// TIA Portal project "Esercizio_contatore" (V15.1)

(* hardware
DEVICE "S7-1200 station_1"  S7-1200 Station
   slot 0: "Telaio di montaggio_0"  S7-1200 Rack  Rack  V1.0
   slot 1: "PLC_1"  CPU 1214C DC/DC/DC  6ES7 214-1AG40-0XB0  V4.2
*)

// ===== PLC "PLC_1"  CPU 1214C DC/DC/DC =====

VAR_GLOBAL CONSTANT   // PLC tag table "Tabella delle variabili standard"
   "valoreMassimo" : Int := 10;
END_VAR

DATA_BLOCK "blocco dati"   // DB1
{ S7_Optimized_Access := 'TRUE' }
VERSION : 0.1
   VAR RETAIN
      "A" : Array[0..9] of Int;
      contatore : Int;
   END_VAR
BEGIN
END_DATA_BLOCK

ORGANIZATION_BLOCK "Main"   // OB1, LAD, ProgramCycle
TITLE = "Main Program Sweep (Cycle)"
{ S7_Optimized_Access := 'TRUE' }
VERSION : 0.1
   VAR_INPUT
      Initial_Call : Bool;   // Initial call of this OB
      Remanence : Bool;   // =True, if remanent data are available
   END_VAR
BEGIN
END_ORGANIZATION_BLOCK

ORGANIZATION_BLOCK "Cyclic interrupt"   // OB30, LAD, CyclicInterrupt
{ S7_Optimized_Access := 'TRUE' }
VERSION : 0.1
   VAR_INPUT
      Initial_Call : Bool;   // Initial call of this OB
      Event_Count : Int;   // Events discarded
   END_VAR
BEGIN

REGION Network 1
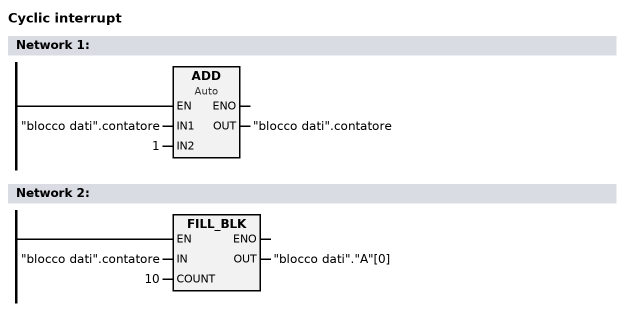
   RUNG wire#powerrail
      Add(in1 := "blocco dati".contatore, in2 := 1, out => "blocco dati".contatore)
   END_RUNG
   // the same network as SCL:
   "blocco dati".contatore := "blocco dati".contatore + 1;
END_REGION

REGION Network 2
   RUNG wire#powerrail
      FillBlockI(in := "blocco dati".contatore, count := 10, out => "blocco dati"."A"[0])
   END_RUNG
   // the same network as SCL:
   FILL_BLK(IN := "blocco dati".contatore, COUNT := 10, OUT => "blocco dati"."A"[0]);
END_REGION
END_ORGANIZATION_BLOCK